TYPE ST_Reminders :
STRUCT
	bSolventLevels 		: BOOL := FALSE;
	bWasteLevel			: BOOL := FALSE;
	bVialRackPresent	: BOOL := FALSE;
	bRecipeActivated	: BOOL := FALSE;
	bThroatJigPresent	: BOOL := FALSE;
	bAutoCicleReady		: BOOL := FALSE;
	bStagePlateHomePos	: BOOL := FALSE;
	bVialRackRemoved	: BOOL := FALSE;
	bCalBoxInPlace		: BOOL := FALSE;
	bCalibrationReady	: BOOL := FALSE;
END_STRUCT
END_TYPE

(* stored: Version 1.1.0.1, ProductVersion 3.1.4024.15
   DUT ST_Reminders: Id {099df7a4-2817-41f2-8bfb-53dab4de2f12} *)
